FUNCTION_BLOCK FB_HeatpumpIO
VAR_OUTPUT
	stProcessData 		: 	ST_ProcessData;
END_VAR
VAR
END_VAR


IO.bOutputN1 := IO.bInputN1;

END_FUNCTION_BLOCK

(* stored: Version 1.1.0.1
   POU FB_HeatpumpIO: Id {97d548f3-37ea-4aba-ae88-86175ac4851e}, SpecialFunc None *)
